FUNCTION MA_Jump : INT

VAR_INPUT
	//Enable: BOOL:=0;
	Speed: REAL:=0;
	Bump_Duration: TIME:=T#0MS;
	//Bump_Trigger: BOOL := 0;
END_VAR


VAR_IN_OUT
	Axis: Motion_Axis;
END_VAR

VAR
	i: INT:=0;
END_VAR

Axis.IN_Closed_Open_Loop:=0;
Axis.IN_Enable_Control:=1;
Axis.OL_IN_Analog:=Speed;
Axis.OL_IN_Slave_Enable:=0;
Axis.OL_Move_Type:=1;
Axis.OL_IN_Bump_Duration:= Bump_Duration;  //Timer for Bump Type of Move
Axis.OL_IN_Bump_Trigger:= 1;

END_FUNCTION

(* stored: Version 1.1.0.1, ProductVersion 3.1.4020.12
   POU MA_Jump: Id {1532186e-e2ed-4daf-805b-0019b866528b}, SpecialFunc None *)
